DATA_BLOCK "Station7LoadData"
{ S7_Optimized_Access := 'FALSE' }
VERSION : 0.1
NON_RETAIN
   STRUCT
      "PLC.PartTypeID" : Int;
      "PLC.Station7RecipeNo" : Int;
      "PLC.Station7DMXCode" : String[128];
      "PLC.SubPartSN1" : String[128];
      "MES.ErrorCode" : Int;
      "MES.StatusBits" : DInt;
      "MES.Cycle_ID" : DInt;
      "MES.Unit_ParttypeID" : Int;
   END_STRUCT;


BEGIN

END_DATA_BLOCK

